{attribute 'qualified_only'}
{attribute 'strict'}
TYPE eDcInputType :
(
	None := 0,
	Dc_charger := 1, 
	Dc_extender := 2
);
END_TYPE

(* stored: Version 1.1.0.1, ProductVersion 3.1.4026.18
   DUT eDcInputType: Id {7bdbb057-36f4-4580-9758-e9ac5c99603a} *)
